PROGRAM MAIN
VAR
	bDummt : BOOL;
END_VAR

END_PROGRAM

(* stored: Version 1.1.0.1, ProductVersion 3.1.4024.12
   POU MAIN: Id {dec0af98-17e5-408d-9a84-a18f5a03faac}, SpecialFunc None *)
